// TIA Portal V17 export
// export: Created 2024-10-17T14:16:17.0939194Z, ExportSetting WithDefaults, DisplayName Totally Integrated Automation Portal, DisplayVersion V17 Update 4, DisplayName TIA Portal Openness, DisplayVersion V17 Update 4, DisplayName TIA Portal Version Control Interface, DisplayVersion V17, DisplayName SINAMICS Startdrive Advanced, DisplayVersion V17 Update2, DisplayName SINAMICS Startdrive G130, G150, S120, S150, SINAMICS MV, S210, DisplayVersion V17 Update2, DisplayName SINAMICS Startdrive G110M, G120, G120C, G120D, G120P, G115D, DisplayVersion V17 Update2, DisplayName STEP 7 Professional, DisplayVersion V17 Update 4, DisplayName STEP 7 Safety, DisplayVersion V17, DisplayName WinCC Advanced / Unified PC, DisplayVersion V17 Update 4
TYPE "LPMLV2022_typeCommand"
TITLE = LPMLV2022_typeCommand
// Support: tech.team.motioncontrol@siemens.com
// stored: IsFailsafeCompliant false
   STRUCT
      UnitMode : DInt;   // Unit Mode Target (0: Invalid, 1: Production, 2: Maintenance, 3: Manual, 04 - 31: User Definable). Minimum required for supervisory control
      UnitModeChangeRequest : Bool;   // Request Unit Mode Change to Unit Mode Target. Minimum required for supervisory control
      MachSpeed : Real;   // Current Machine Speed Setpoint; Unit of Measure: Primary Packages/Minute. Minimum required for supervisory control
      MaterialInterlock : DWord;   // Materials Ready. It is comprised of a series of bits with 1 equaling ready or not low, 0 equaling not ready, or low. Each bit represents a different user material. Unused bits should be forced to a value of 1 or TRUE
      CntrlCmd : DInt;   // Control Command (0: Undefined, 1: Reset, 2: Start, 3: Stop, 4: Hold, 5: UnHold, 6: Suspend, 7: UnSuspend, 8: Abort, 9: Clear, 10: Complete). Minimum required for supervisory control
      CmdChangeRequest : Bool;   // State Change Request. This CmdChangeRequest bit will command the machine to proceed to change the state to the target state. Minimum required for supervisory control
      Parameter_REAL : Array[0.."LPMLV2022_COMMAND_PARAMETER_REAL_UPPER_LIM"] of "LPMLV2022_typeParameter_REAL";   // Structured Array of Unit/Machine Parameter information for values with REAL data type
      Parameter_STRING : Array[0.."LPMLV2022_COMMAND_PARAMETER_STRING_UPPER_LIM"] of "LPMLV2022_typeParameter_STRING";   // Structured Array of Unit/Machine Parameter information for values with STRING data type
      Parameter_LREAL : Array[0.."LPMLV2022_COMMAND_PARAMETER_LREAL_UPPER_LIM"] of "LPMLV2022_typeParameter_LREAL";   // Structured Array of Unit/Machine Parameter information for values with LREAL data type
      Parameter_DINT : Array[0.."LPMLV2022_COMMAND_PARAMETER_DINT_UPPER_LIM"] of "LPMLV2022_typeParameter_DINT";   // Structured Array of Unit/Machine Parameter information for values with DINT data type
      Parameter_BOOL : Array[0.."LPMLV2022_COMMAND_PARAMETER_BOOL_UPPER_LIM"] of "LPMLV2022_typeParameter_BOOL";   // Structured Array of Unit/Machine Parameter information for values with BOOL data type
      SelectedRecipe : DInt;   // Recipe Selection. This tag is used to designate which recipe should be run on the machine to produce the primary output product, according to a user-design recipe handling procedure. It is designed to correspond directly to the listing in the Recipe Array
      RecipeChangeRequest : Bool;   // Recipe change request. This tag is used to trigger a user-defined recipe changeover process that will configure the machine to produce the primary product designated in Command.SelectedRecipe
      Recipe : Array[0.."LPMLV2022_COMMAND_RECIPE_UPPER_LIM"] of "LPMLV2022_typeCommandRecipe";   // Structured Array of Recipe Information. The recipe data type can be used for defining product ingredient and product processing parameter variables
   END_STRUCT;
END_TYPE
